// TIA Portal V15 export
// export: Created 2019-02-22T09:02:39.5689267Z, ExportSetting WithDefaults, WithReadOnly, DisplayName Totally Integrated Automation Portal, DisplayVersion V15 Update 2, DisplayName TIA Portal Openness, DisplayVersion V15 Update 2, DisplayName STEP 7 Professional, DisplayVersion V15 Update 2, DisplayName STEP 7 Safety, DisplayVersion V15, DisplayName WinCC Professional, DisplayVersion V15 Update 2, DisplayName SIMATIC Visualization Architect, DisplayVersion V15 Update 1
DATA_BLOCK "FGDB_STATION_NAME"   // DB155
TITLE = Station STATION_NR / Station 010
{ S7_Optimized_Access := 'FALSE' }
AUTHOR : integra
FAMILY : BS
VERSION : 0.5
// stored: AutoNumber true, CodeModifiedDate 2018-10-17T05:47:33.8335142Z, CompileDate 2019-01-06T16:25:47.51981Z, CreationDate 2018-11-16T09:32:53.5033139Z, DBAccessibleFromOPCUA true, InstanceOfName iFG_STATION, InstanceOfNumber 1019, InstanceOfType FB, InterfaceModifiedDate 2018-01-24T11:37:23.2619932Z, IsConsistent true, IsKnowHowProtected false, ModifiedDate 2018-10-17T05:47:33.8335142Z, ParameterModified 2016-03-08T16:45:31.2607837Z, StructureModified 2016-10-24T09:10:27.3679338Z, UDAEnableTagReadback false
"iFG_STATION"
   // VAR_INPUT
   //    station : Int;
   //    fct : Int;
   //    initialPos : Bool;
   // END_VAR
   // VAR_OUTPUT
   //    fault : Bool;
   //    faultExt : Bool;
   // END_VAR
   // VAR RETAIN
   //    idx : Int;
   //    sectionNumber : Int;
   //    deskNumber : Int;
   //    stationNumber : Int;
   //    dbNumber : Int;
   //    function : Int;
   //    numberInternalMessages : Int;
   //    numberExternalMessages : Int;
   //    F : Struct
   //       fct : Bool;
   //    END_STRUCT;
   //    Masks : Struct
   //       disableFault_1_8 : Byte;
   //       prodRelevantFault_1_8 : Byte;
   //    END_STRUCT;
   //    LastState : Struct
   //       fault_1_8 : Byte;
   //    END_STRUCT;
   //    IfcFGExternal : "iUDT_IFC_SYS_EXTERNAL_ALARM";
   //    ExtP : Struct
   //       setup : Bool;
   //       auto : Bool;
   //       enableIn : Bool;
   //       ack : Bool;
   //    END_STRUCT;
   //    StM : Struct
   //       fault : Bool;
   //       setup : Bool;
   //       auto : Bool;
   //       warning : Bool;
   //       eStop : Bool;
   //       safetyStop : Bool;
   //       enableIn : Bool;
   //       enableOutForward : Bool;
   //       enableOutBackward : Bool;
   //       faultPr : Bool;
   //       pairMon : Bool;
   //       specialMode : Bool;
   //       "13" : Bool;
   //       "14" : Bool;
   //       "15" : Bool;
   //       "16" : Bool;
   //       "17" : Bool;
   //       "18" : Bool;
   //       "19" : Bool;
   //       "20" : Bool;
   //       "21" : Bool;
   //       "22" : Bool;
   //       "23" : Bool;
   //       "24" : Bool;
   //       "25" : Bool;
   //       "26" : Bool;
   //       "27" : Bool;
   //       "28" : Bool;
   //       "29" : Bool;
   //       "30" : Bool;
   //       "31" : Bool;
   //       "32" : Bool;
   //    END_STRUCT;
   //    VB : Struct
   //       fault : Bool;
   //       setup : Bool;
   //       auto : Bool;
   //       warning : Bool;
   //       eStop : Bool;
   //       safetyStop : Bool;
   //       enableIn : Bool;
   //       enableOutForward : Bool;
   //       enableOutBackward : Bool;
   //       faultPr : Bool;
   //       pairMon : Bool;
   //       specialMode : Bool;
   //       "13" : Bool;
   //       "14" : Bool;
   //       "15" : Bool;
   //       "16" : Bool;
   //       "17" : Bool;
   //       "18" : Bool;
   //       "19" : Bool;
   //       "20" : Bool;
   //       "21" : Bool;
   //       "22" : Bool;
   //       "23" : Bool;
   //       "24" : Bool;
   //       "25" : Bool;
   //       "26" : Bool;
   //       "27" : Bool;
   //       "28" : Bool;
   //       "29" : Bool;
   //       "30" : Bool;
   //       "31" : Bool;
   //       "32" : Bool;
   //    END_STRUCT;
   //    VCB : Struct
   //       ack : Bool;
   //    END_STRUCT;
   //    D : Struct
   //       visuAck : Bool;
   //       enableln : Bool;
   //       initialPos : Bool;
   //    END_STRUCT;
   //    V : Struct
   //       runtime : UInt;
   //    END_STRUCT;
   // END_VAR
BEGIN
END_DATA_BLOCK
